FUNCTION_BLOCK ExecuteBase EXTENDS CommonBase
VAR_INPUT
END_VAR
VAR_OUTPUT
END_VAR
VAR
END_VAR

METHOD Execute : BOOL
VAR_INPUT
	argCommand : eCylinderCommands;
END_VAR
END_METHOD

END_FUNCTION_BLOCK

(* stored: Version 1.1.0.1, ProductVersion 3.1.4024.0
   POU ExecuteBase: Id {31f85d56-6d2b-43f6-82c0-18b487d86a3e}, SpecialFunc None
   Method Execute: Id {947e425d-0a86-42d4-a40b-e9e1ca16f7ae} *)
